FUNCTION sub_mat : BOOL
VAR_IN_OUT
	a:ARRAY[*,*] OF LREAL;
	b:ARRAY[*,*] OF LREAL;
	c:ARRAY[*,*] OF LREAL;


END_VAR
VAR_INPUT
		m,n:SINT;
END_VAR
VAR_OUTPUT
END_VAR
VAR
	i,j:int;
END_VAR

    FOR i:=0 TO m DO
        FOR j:=0TO n DO
            c[i,j] := a[i,j]-b[i,j];
			END_FOR
			END_FOR
			sub_mat:=true;

END_FUNCTION

(* stored: Version 1.1.0.1, ProductVersion 3.1.4024.12
   POU sub_mat: Id {853f38ee-a0c3-4de3-b2a5-a6fb0ac4e4e0}, SpecialFunc None *)
